{attribute 'linkalways'}
{attribute 'no_explicit_call' := 'This FB is a CLASS and must be accessed using methods or properties'}
FUNCTION_BLOCK PUBLIC AdsLogTargetAdapter IMPLEMENTS LogTargetAdapter
VAR
	formatter : DefaultAdsLogEventFormatter;
END_VAR

METHOD PUBLIC Run
// Do nothing for this, as it directly logs
END_METHOD

METHOD PUBLIC SendLogEvent : BOOL
VAR_INPUT
	event : LogEvent;
END_VAR
Tc2_System.AdsLogStr(
	AdsLog_MsgType_Log OR LogLevelToAdsLogMsgType(event.level), 
	formatter.Format(event), 
	''
);
END_METHOD

END_FUNCTION_BLOCK

(* stored: Version 1.1.0.1
   POU AdsLogTargetAdapter: Id {416ec712-fa42-449e-b7e8-011b9755b87d}, SpecialFunc None
   Method Run: Id {87c612cd-8012-4f19-95eb-e105b1ccb4db}
   Method SendLogEvent: Id {3e9a19fd-876a-41d8-81fb-3daddc75cd4b} *)
